{attribute 'Tc2GvlVarNames'}
VAR_GLOBAL
	iDeviceTasterVisu			:INT := 1;
	iDeviceRelaisVisu			:INT := cMaxBusTaster+1;
	iDeviceCYDVisu				:INT := cMaxBusTaster+cMaxBusRelais+1;
	
	bTasterServiceAktiv			:ARRAY[1..cMaxBusTaster] OF BOOL;
	bRelaisServiceAktiv			:ARRAY[cMaxBusTaster+1..cMaxBusTaster+cMaxBusRelais+1] OF BOOL;
	bCYDServiceAktiv			:ARRAY[cMaxBusRelais+cMaxBusTaster+2..cMaxBusRelais+cMaxBusTaster+cMaxCYD+1] OF BOOL;
	
	stTasterService				:ARRAY[1..cMaxBusTaster] OF ST_BusTaster6F_Input;
	stRelaisService				:ARRAY[cMaxBusTaster+1..cMaxBusTaster+cMaxBusRelais+1] OF ST_BusRelais16F_Input;
	stCYDService				:ARRAY[cMaxBusRelais+cMaxBusTaster+2..cMaxBusRelais+cMaxBusTaster+cMaxCYD+1] OF ST_BusCYD6F_Input;
END_VAR

(* stored: Version 1.1.0.1, ProductVersion 3.1.4024.12
   GVL GVL_ServiceVisu_1: Id {3cfa0c52-753a-4159-a39b-08a53f1554b7} *)
